{attribute 'GeneratedUsingTerminal: EPP2339-0021-0016'}
{attribute addProperty BoxType "EPP2339-0021-0016"}
{attribute addProperty Id "OutputAT %Q*BOOL1"}
{attribute addProperty CRC "1120571895"}
{attribute addProperty Size "1"}
TYPE Channel_42CA91F7 EXTENDS DigitalOutputBase_1FE0D5EE :
STRUCT
	{attribute addProperty Name "Output"}
	Output AT %Q* : BOOL;
END_STRUCT
END_TYPE

(* stored: Version 1.2.0.0, ProductVersion 3.1.4024.9
   DUT Channel_42CA91F7: Id {dc3a3eec-c31a-4903-9f4d-23cdc31cc7b2} *)
